(* CoDeSys 2.3.9.40 project: мдвв.pro *)
(* Libraries: STANDARD.LIB 4.10.05 11:14:46, IECSFC.LIB 13.4.06 15:51:28, SYSLIBTIME.LIB 20.2.06 13:31:16, SYSTASKINFO.LIB 20.2.06 13:31:38, ANALYZATION.LIB 5.10.99 09:05:06, SYSLIBCALLBACK.LIB 20.2.06 13:31:08 *)

(* PLC configuration (modules and I/O channels)
Discrete input 6 bit [ID100] node 0, in %IB0 out %QB0 {Filtrationtime = 10; Filtrationtime = 10; Filtrationtime = 10; Filtrationtime = 10; Filtrationtime = 10; Filtrationtime = 10; Visibility = No; PinCount = 6; WatchDogPeriod = 1000; PollPeriod = 1}
  AT %IX0.0 [BitInput]
  AT %IX0.1 [BitInput]
  AT %IX0.2 [BitInput]
  AT %IX0.3 [BitInput]
  AT %IX0.4 [BitInput]
  AT %IX0.5 [BitInput]
Discrete output 4 bit [ID101] node 1, in %IB1 out %QB1 {PinCount = 4; SafeValueBool = FALSE; SafeValueBool = FALSE; SafeValueBool = FALSE; SafeValueBool = FALSE; Visibility = No}
  AT %QX1.0 [BitOutput]
  AT %QX1.1 [BitOutput]
  AT %QX1.2 [BitOutput]
  AT %QX1.3 [BitOutput]
Special output [ID104] node 2, in %IB2 out %QB2 {Visibility = No; PinCount = 1}
  AT %QX2.0 [BitOutput] Special output
Unifed signal sensor [ID700] node 3, in %IB3 out %QB3 {Type_of_sensor700 = IT_0_20; measure_interval = 0.8; ainlow = 0; ainhigh = 20; first_cor_point = 0; first_delta = 0; second_cor_point = 0; second_delta = 0; third_cor_point = 0; third_delta = 0; Visibility = No}
  AT %ID3.0 [FloatInput] Value
  AT %IW3.1 [WordInput] Circular time
  Analog Input [ID107] node 0, in %IB3.0 out %QB3.0
Unifed signal sensor [ID700] node 4, in %IB4 out %QB4 {Type_of_sensor700 = IT_0_20; measure_interval = 0.8; ainlow = 0; ainhigh = 20; first_cor_point = 0; first_delta = 0; second_cor_point = 0; second_delta = 0; third_cor_point = 0; third_delta = 0; Visibility = No}
  AT %ID4.0 [FloatInput] Value
  AT %IW4.1 [WordInput] Circular time
  Analog Input [ID107] node 0, in %IB4.0 out %QB4.0
Unifed signal sensor [ID700] node 5, in %IB5 out %QB5 {Type_of_sensor700 = IT_0_20; measure_interval = 0.8; ainlow = 0; ainhigh = 20; first_cor_point = 0; first_delta = 0; second_cor_point = 0; second_delta = 0; third_cor_point = 0; third_delta = 0; Visibility = No}
  AT %ID5.0 [FloatInput] Value
  AT %IW5.1 [WordInput] Circular time
  Analog Input [ID107] node 0, in %IB5.0 out %QB5.0
Unifed signal sensor [ID700] node 6, in %IB6 out %QB6 {Type_of_sensor700 = IT_0_20; measure_interval = 0.8; ainlow = 0; ainhigh = 20; first_cor_point = 0; first_delta = 0; second_cor_point = 0; second_delta = 0; third_cor_point = 0; third_delta = 0; Visibility = No}
  AT %ID6.0 [FloatInput] Value
  AT %IW6.1 [WordInput] Circular time
  Analog Input [ID107] node 0, in %IB6.0 out %QB6.0
Analog output [ID106] node 7, in %IB7 out %QB7 {DAC_Type = Voltage 0-10 B; Analog_offset_correction = 0; Analog_full_range_correction = 0; SafeValueFloat = 0; Visibility = No}
  AT %QD7.0 [FloatOutput] Value
Analog output [ID106] node 8, in %IB8 out %QB8 {DAC_Type = Voltage 0-10 B; Analog_offset_correction = 0; Analog_full_range_correction = 0; SafeValueFloat = 0; Visibility = No}
  AT %QD8.0 [FloatOutput] Value
AT %QD9.0 [DWordOutput] Last address
AT %QW9.1 [WordOutput] Last error
RS-485-1 [COM1_USART] node 0, in %IB9.0 out %QB9.0 {CommunicationSpeed = 9600; Parity = NO PARITY CHECK; BitLength = 8 bits; StopLength = One stop bit; InterfaceType = RS485; FrameOriented = RTU; Timeout = 0; Visibility = No}
AT %QB9.1.0 [ComChannel] Command (0xff - Start)
Value on Output ¹1 [ID2098] node 0, in %IB9.1.0 out %QB9.1.0 {ModbusAddress = 0; Comm_Write_16 = Command Write (16); Visibility = No}
  AT %QW9.1.0.0 [WordOutput]
Value on Output ¹2 [ID2099] node 1, in %IB9.1.1 out %QB9.1.1 {ModbusAddress = 1; Comm_Write_16 = Command Write (16); Visibility = No}
  AT %QW9.1.1.0 [WordOutput]
Value on Output ¹3 [ID2150] node 2, in %IB9.1.2 out %QB9.1.2 {ModbusAddress = 2; Comm_Write_16 = Command Write (16); Visibility = No}
  AT %QW9.1.2.0 [WordOutput]
Value on Output ¹4 [ID2151] node 3, in %IB9.1.3 out %QB9.1.3 {ModbusAddress = 3; Comm_Write_16 = Command Write (16); Visibility = No}
  AT %QW9.1.3.0 [WordOutput]
Value on Output ¹5 [ID2152] node 4, in %IB9.1.4 out %QB9.1.4 {ModbusAddress = 4; Comm_Write_16 = Command Write (16); Visibility = No}
  AT %QW9.1.4.0 [WordOutput]
Value on Output ¹6 [ID2153] node 5, in %IB9.1.5 out %QB9.1.5 {ModbusAddress = 5; Comm_Write_16 = Command Write (16); Visibility = No}
  AT %QW9.1.5.0 [WordOutput]
Value on Output ¹7 [ID2154] node 6, in %IB9.1.6 out %QB9.1.6 {ModbusAddress = 6; Comm_Write_16 = Command Write (16); Visibility = No}
  AT %QW9.1.6.0 [WordOutput]
Value on Output ¹8 [ID2155] node 7, in %IB9.1.7 out %QB9.1.7 {ModbusAddress = 7; Comm_Write_16 = Command Write (16); Visibility = No}
  AT %QW9.1.7.0 [WordOutput]
PWM period on Output ¹1 [ID2156] node 8, in %IB9.1.8 out %QB9.1.8 {ModbusAddress = 32; Comm_Write_16 = Command Write (16); Visibility = No}
  AT %QW9.1.8.0 [WordOutput]
  AT %QB9.1.8.1 [ComChannel] Command (0xff - Start)
PWM period on Output ¹2 [ID2157] node 9, in %IB9.1.9 out %QB9.1.9 {ModbusAddress = 33; Comm_Write_16 = Command Write (16); Visibility = No}
  AT %QW9.1.9.0 [WordOutput]
  AT %QB9.1.9.1 [ComChannel] Command (0xff - Start)
PWM period on Output ¹3 [ID2158] node 10, in %IB9.1.10 out %QB9.1.10 {ModbusAddress = 34; Comm_Write_16 = Command Write (16); Visibility = No}
  AT %QW9.1.10.0 [WordOutput]
  AT %QB9.1.10.1 [ComChannel] Command (0xff - Start)
PWM period on Output ¹4 [ID2159] node 11, in %IB9.1.11 out %QB9.1.11 {ModbusAddress = 35; Comm_Write_16 = Command Write (16); Visibility = No}
  AT %QW9.1.11.0 [WordOutput]
  AT %QB9.1.11.1 [ComChannel] Command (0xff - Start)
PWM period on Output ¹5 [ID2160] node 12, in %IB9.1.12 out %QB9.1.12 {ModbusAddress = 36; Comm_Write_16 = Command Write (16); Visibility = No}
  AT %QW9.1.12.0 [WordOutput]
  AT %QB9.1.12.1 [ComChannel] Command (0xff - Start)
PWM period on Output ¹6 [ID2161] node 13, in %IB9.1.13 out %QB9.1.13 {ModbusAddress = 37; Comm_Write_16 = Command Write (16); Visibility = No}
  AT %QW9.1.13.0 [WordOutput]
  AT %QB9.1.13.1 [ComChannel] Command (0xff - Start)
PWM period on Output ¹7 [ID2162] node 14, in %IB9.1.14 out %QB9.1.14 {ModbusAddress = 38; Comm_Write_16 = Command Write (16); Visibility = No}
  AT %QW9.1.14.0 [WordOutput]
  AT %QB9.1.14.1 [ComChannel] Command (0xff - Start)
PWM period on Output ¹8 [ID2163] node 15, in %IB9.1.15 out %QB9.1.15 {ModbusAddress = 39; Comm_Write_16 = Command Write (16); Visibility = No}
  AT %QW9.1.15.0 [WordOutput]
  AT %QB9.1.15.1 [ComChannel] Command (0xff - Start)
Bit Mask for output [ID2164] node 16, in %IB9.1.16 out %QB9.1.16 {ModbusAddress = 50; Comm_Write_16 = Command Write (16); Visibility = No}
  AT %QW9.1.16.0 [WordOutput]
  AT %QB9.1.16.1 [ComChannel] Command (0xff - Start)
Bit Mask for input [ID2165] node 17, in %IB9.1.17 out %QB9.1.17 {ModbusAddress = 51; Comm_Read_03 = Command Read (03); Visibility = No}
  AT %IW9.1.17.0 [WordInput]
Value of input counter ¹1 [ID2166] node 18, in %IB9.1.18 out %QB9.1.18 {ModbusAddress = 64; Comm_Read_03 = Command Read (03); Visibility = No}
  AT %IW9.1.18.0 [WordInput]
Value of input counter ¹2 [ID2167] node 19, in %IB9.1.19 out %QB9.1.19 {ModbusAddress = 65; Comm_Read_03 = Command Read (03); Visibility = No}
  AT %IW9.1.19.0 [WordInput]
Value of input counter ¹3 [ID2168] node 20, in %IB9.1.20 out %QB9.1.20 {ModbusAddress = 66; Comm_Read_03 = Command Read (03); Visibility = No}
  AT %IW9.1.20.0 [WordInput]
Value of input counter ¹4 [ID2169] node 21, in %IB9.1.21 out %QB9.1.21 {ModbusAddress = 67; Comm_Read_03 = Command Read (03); Visibility = No}
  AT %IW9.1.21.0 [WordInput]
Value of input counter ¹5 [ID2170] node 22, in %IB9.1.22 out %QB9.1.22 {ModbusAddress = 68; Comm_Read_03 = Command Read (03); Visibility = No}
  AT %IW9.1.22.0 [WordInput]
Value of input counter ¹6 [ID2171] node 23, in %IB9.1.23 out %QB9.1.23 {ModbusAddress = 69; Comm_Read_03 = Command Read (03); Visibility = No}
  AT %IW9.1.23.0 [WordInput]
Value of input counter ¹7 [ID2172] node 24, in %IB9.1.24 out %QB9.1.24 {ModbusAddress = 70; Comm_Read_03 = Command Read (03); Visibility = No}
  AT %IW9.1.24.0 [WordInput]
Value of input counter ¹8 [ID2173] node 25, in %IB9.1.25 out %QB9.1.25 {ModbusAddress = 71; Comm_Read_03 = Command Read (03); Visibility = No}
  AT %IW9.1.25.0 [WordInput]
Value of input counter ¹9 [ID2174] node 26, in %IB9.1.26 out %QB9.1.26 {ModbusAddress = 72; Comm_Read_03 = Command Read (03); Visibility = No}
  AT %IW9.1.26.0 [WordInput]
Value of input counter ¹10 [ID2175] node 27, in %IB9.1.27 out %QB9.1.27 {ModbusAddress = 73; Comm_Read_03 = Command Read (03); Visibility = No}
  AT %IW9.1.27.0 [WordInput]
Value of input counter ¹11 [ID2176] node 28, in %IB9.1.28 out %QB9.1.28 {ModbusAddress = 74; Comm_Read_03 = Command Read (03); Visibility = No}
  AT %IW9.1.28.0 [WordInput]
Value of input counter ¹12 [ID2177] node 29, in %IB9.1.29 out %QB9.1.29 {ModbusAddress = 75; Comm_Read_03 = Command Read (03); Visibility = No}
  AT %IW9.1.29.0 [WordInput]
*)

(* POU PLC_PRG, CFC *)
PROGRAM PLC_PRG
VAR
END_VAR
_CFC_ (* Continuous Function Chart, elements in execution order *)
_END_CFC_
END_PROGRAM
